# EPICS autosave request: apps/svtIntlkApp/Db/svtIntlk.req
#
# SVT Soft Interlock settings
#
$(P)intlk_delay
$(P)min
$(P)max
$(P)intlk_bypass
$(P)intlk_reset
$(P)intlk_status
